// TIA Portal V21 export
TYPE "stopCtxHMI"
   STRUCT
      "step" : USInt;
      stepTime : LTime;
      alm { S7_SetPoint := 'True'} : DWord;
   END_STRUCT;
END_TYPE
